{attribute 'qualified_only'}
{attribute 'strict'}
TYPE E_FeatureScalingType :
(
	NONE := 0,
	MAXABS,
	MINMAX,
	MINMAX_EXP,
	STANDARDIZATION,
	CUSTOM
);
END_TYPE

(* stored: Version 1.1.0.1, ProductVersion 3.1.4024.12
   DUT E_FeatureScalingType: Id {d7983fcd-8a7f-429c-9076-91467d4f6eeb} *)
